// ARGB component builder.
FUNCTION_BLOCK Argbb
VAR
	_r: BYTE;
	_g: BYTE;
	_b: BYTE;
	_a: BYTE;
END_VAR

// Alpha channel.
PROPERTY Alpha : BYTE
GET
Alpha := _a;
END_GET
SET
_a := Alpha;
END_SET
END_PROPERTY

// Blue channel.
PROPERTY Blue : BYTE
GET
Blue := _b;
END_GET
SET
_b := Blue;
END_SET
END_PROPERTY

// Green channel.
PROPERTY Green : BYTE
GET
Green := _g;
END_GET
SET
_g := Green;
END_SET
END_PROPERTY

// Packed ARGB value.
PROPERTY Raw : Argb
GET
Raw := 	USINT_TO_UDINT(_b) OR
			SHL(USINT_TO_UDINT(_g), 8) OR
			SHL(USINT_TO_UDINT(_r), 16) OR
			SHL(USINT_TO_UDINT(_a), 24);
END_GET
SET
_b := UDINT_TO_USINT(Raw AND 16#FF);
_g := UDINT_TO_USINT(SHR(Raw, 8) AND 16#FF);
_r := UDINT_TO_USINT(SHR(Raw, 16) AND 16#FF);
_a := UDINT_TO_USINT(SHR(Raw, 24) AND 16#FF);
END_SET
END_PROPERTY

// Red channel.
PROPERTY Red : BYTE
GET
Red := _r;
END_GET
SET
_r := Red;
END_SET
END_PROPERTY

// Sets all color channels.
METHOD Set
VAR_INPUT
	nRed: USINT; // Red channel.
	nGreen: USINT; // Green channel.
	nBlue: USINT; // Blue channel.
	nAlpha: USINT; // Alpha channel.
END_VAR
_r := nRed;
_g := nGreen;
_b := nBlue;
_a := nAlpha;
END_METHOD

END_FUNCTION_BLOCK

(* stored: Version 1.1.0.1
   POU Argbb: Id {d884fe8f-dddb-49ad-9aef-a4f440a46ea0}, SpecialFunc None
   Property Alpha: Id {ee2a864b-72ce-497e-8860-76928872cda1}
   Get Get: Id {6604ddfc-f720-4321-9d50-1c51f2738342}
   Set Set: Id {22ca581c-eeff-42f7-b89c-3d4fffd7dfb4}
   Property Blue: Id {3f1ac743-1c2b-4d63-bdad-2ec08f81e45a}
   Get Get: Id {c4a3c42c-2203-4d76-8c0a-3bc8fb749fb9}
   Set Set: Id {9cb8ecae-c8ec-4c3b-b497-9d90de0cfbf2}
   Property Green: Id {34fb47af-42ff-4bce-9fe5-a581493cffea}
   Get Get: Id {73b3330f-5972-409a-b6b3-22231de1acf8}
   Set Set: Id {f0abe708-c83e-4ada-a9f3-b098a0382609}
   Property Raw: Id {7498ed64-bd4c-4ff5-82e1-2e5e41239c2d}
   Get Get: Id {7bd33e5f-4efa-455b-8c3e-295fca724c53}
   Set Set: Id {115bbdd4-d73f-4b8e-8f6c-e1130736bd89}
   Property Red: Id {96853ed3-5cc1-41dc-ad25-9f66e3e7fc3b}
   Get Get: Id {91eb7c2b-4415-486f-8050-84a0112e4cbe}
   Set Set: Id {4dbbf1ab-b554-4ee9-80e6-1892940e1800}
   Method Set: Id {de1e52bc-10d3-4d8a-8f2c-41becbc12b53} *)
